PROGRAM AchtB
VAR
	Woonruimte			: FB_Gelijkvloers;
	Tuin				: FB_Tuin;
	Slaapkamers			: FB_Slaapkamers;
	Garage				: FB_Garage;
	Technische_ruimte	: FB_Technische_ruimte;
	
END_VAR

PrgMqttCom();

END_PROGRAM

(* stored: Version 1.1.0.1, ProductVersion 3.1.4024.12
   POU AchtB: Id {2e7579de-54ce-4ab9-9603-b3d5b4dc69f3}, SpecialFunc None *)
